// TIA Portal project "Cierre_Centralizado" (V16)

(* hardware
DEVICE "S7-1200 station_1"  S7-1200 Station
   slot 0: "Rack_0"  S7-1200 Rack  Rack  V1.0
   slot 1: "PLC_1"  CPU 1214C AC/DC/Rly  6ES7 214-1BG40-0XB0  V4.2
   slot 3: "AQ 1x12BIT_1"  AQ1 signal board  6ES7 232-4HA30-0XB0  V1.0
*)

// ===== PLC "PLC_1"  CPU 1214C AC/DC/Rly =====

VAR_GLOBAL   // PLC tag table "Entradas"
   "mandoAbrir" AT %I0.0 : Bool;
   "mandoCerrar" AT %I0.1 : Bool;
   "senPC" AT %I0.3 : Bool;
   "senPA" AT %I0.2 : Bool;
   "senVDA" AT %I0.4 : Bool;
   "senVIA" AT %I0.5 : Bool;
   "senVDC" AT %I0.6 : Bool;
   "senVIC" AT %I0.7 : Bool;
END_VAR

VAR_GLOBAL   // PLC tag table "Salidas"
   "releAbrirPuerta" AT %Q0.0 : Bool;
   "releCerrarPuerta" AT %Q0.1 : Bool;
   "releVentanaDerechaAbrir" AT %Q0.2 : Bool;
   "releVentanaIzquierdaAbrir" AT %Q0.3 : Bool;
   "releVentanaDerechaCerrar" AT %Q0.4 : Bool;
   "releVentanaIzquierdaCerrar" AT %Q0.5 : Bool;
END_VAR

VAR_GLOBAL   // PLC tag table "Marcas"
   "mandoAbrir_FA" AT %M6.0 : Bool;
   "mandoCerrar_FA" AT %M6.1 : Bool;
   "mandoCerrar_Aux" AT %M7.1 : Bool;
   "mandoAbrir_Aux" AT %M7.0 : Bool;
END_VAR

DATA_BLOCK "Cierre_Centralizado_DB"   // DB1
{ S7_Optimized_Access := 'TRUE' }
VERSION : 0.1
// stored: InstanceOfName Cierre_Centralizado
"Cierre_Centralizado"
BEGIN
END_DATA_BLOCK

// folder: System blocks/Program resources

DATA_BLOCK "T1"   // DB2
{ S7_Optimized_Access := 'TRUE' }
AUTHOR : Simatic
FAMILY : IEC
NAME : IEC_TMR
VERSION : 1.0
// stored: InstanceOfName IEC_TIMER
"IEC_TIMER"
BEGIN
END_DATA_BLOCK

DATA_BLOCK "T2"   // DB3
{ S7_Optimized_Access := 'TRUE' }
AUTHOR : Simatic
FAMILY : IEC
NAME : IEC_TMR
VERSION : 1.0
// stored: InstanceOfName IEC_TIMER
"IEC_TIMER"
BEGIN
END_DATA_BLOCK

// folder: (top level)

FUNCTION_BLOCK "Cierre_Centralizado"   // FB1, LAD
{ S7_Optimized_Access := 'TRUE' }
VERSION : 0.1
   VAR_INPUT
      Init : Bool := false;
      Reset : Bool;
   END_VAR
   VAR
      X0 : Bool := true;
      X1 : Bool;
      X2 : Bool;
      X3 : Bool;
      X4 : Bool;
      X5 : Bool;
      X6 : Bool;
      X7 : Bool;
      X8 : Bool;
      X9 : Bool;
   END_VAR
BEGIN

REGION Network 1: X0
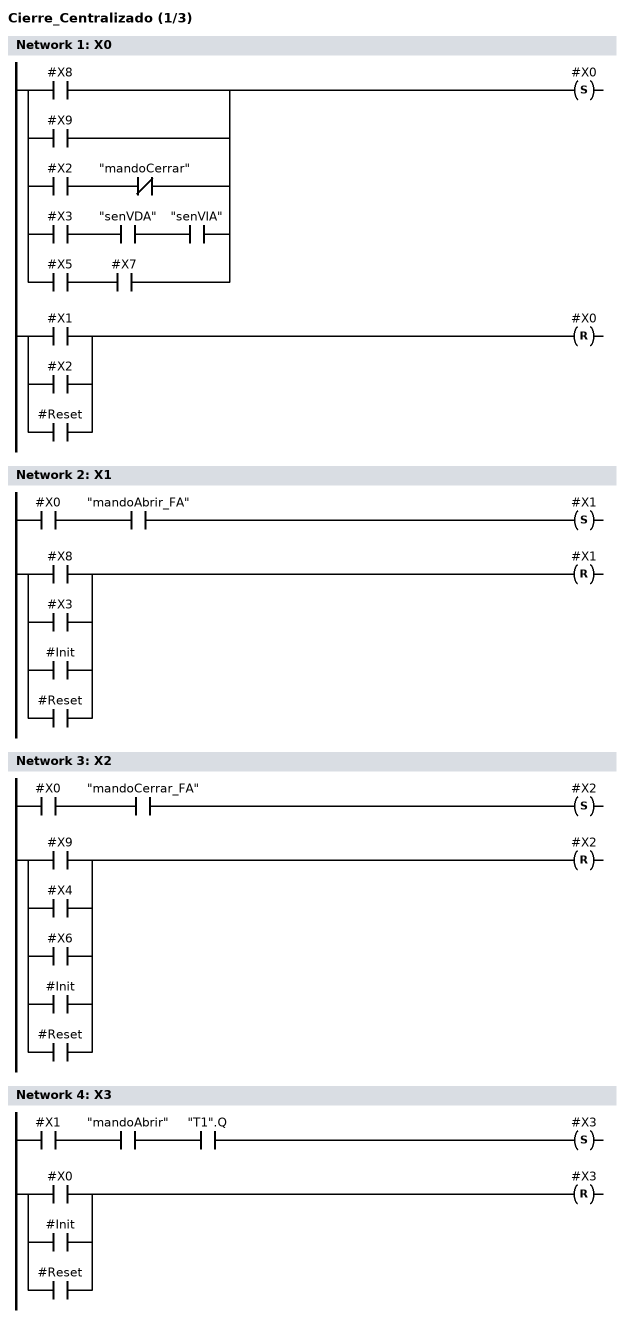
   RUNG wire#powerrail
      Contact( #X8 )
      wire#w1
      S_Coil( #X0 )
   END_RUNG
   RUNG wire#powerrail
      Contact( #X9 )
   END_RUNG wire#w1
   RUNG wire#powerrail
      Contact( #X2 )
      I_Contact( "mandoCerrar" )
   END_RUNG wire#w1
   RUNG wire#powerrail
      Contact( #X3 )
      Contact( "senVDA" )
      Contact( "senVIA" )
   END_RUNG wire#w1
   RUNG wire#powerrail
      Contact( #X5 )
      Contact( #X7 )
   END_RUNG wire#w1
   RUNG wire#powerrail
      Contact( #X1 )
      wire#w2
      R_Coil( #X0 )
   END_RUNG
   RUNG wire#powerrail
      Contact( #X2 )
   END_RUNG wire#w2
   RUNG wire#powerrail
      Contact( #Reset )
   END_RUNG wire#w2
   // the same network as SCL:
   IF #X8 OR #X9 OR (#X2 AND NOT "mandoCerrar") OR (#X3 AND "senVDA" AND "senVIA") OR (#X5 AND #X7) THEN
       #X0 := TRUE;
   END_IF;
   IF #X1 OR #X2 OR #Reset THEN #X0 := FALSE; END_IF;
END_REGION

REGION Network 2: X1
   RUNG wire#powerrail
      Contact( #X0 )
      Contact( "mandoAbrir_FA" )
      S_Coil( #X1 )
   END_RUNG
   RUNG wire#powerrail
      Contact( #X8 )
      wire#w1
      R_Coil( #X1 )
   END_RUNG
   RUNG wire#powerrail
      Contact( #X3 )
   END_RUNG wire#w1
   RUNG wire#powerrail
      Contact( #Init )
   END_RUNG wire#w1
   RUNG wire#powerrail
      Contact( #Reset )
   END_RUNG wire#w1
   // the same network as SCL:
   IF #X0 AND "mandoAbrir_FA" THEN #X1 := TRUE; END_IF;
   IF #X8 OR #X3 OR #Init OR #Reset THEN #X1 := FALSE; END_IF;
END_REGION

REGION Network 3: X2
   RUNG wire#powerrail
      Contact( #X0 )
      Contact( "mandoCerrar_FA" )
      S_Coil( #X2 )
   END_RUNG
   RUNG wire#powerrail
      Contact( #X9 )
      wire#w1
      R_Coil( #X2 )
   END_RUNG
   RUNG wire#powerrail
      Contact( #X4 )
   END_RUNG wire#w1
   RUNG wire#powerrail
      Contact( #X6 )
   END_RUNG wire#w1
   RUNG wire#powerrail
      Contact( #Init )
   END_RUNG wire#w1
   RUNG wire#powerrail
      Contact( #Reset )
   END_RUNG wire#w1
   // the same network as SCL:
   IF #X0 AND "mandoCerrar_FA" THEN #X2 := TRUE; END_IF;
   IF #X9 OR #X4 OR #X6 OR #Init OR #Reset THEN #X2 := FALSE; END_IF;
END_REGION

REGION Network 4: X3
   RUNG wire#powerrail
      Contact( #X1 )
      Contact( "mandoAbrir" )
      Contact( "T1".Q )
      S_Coil( #X3 )
   END_RUNG
   RUNG wire#powerrail
      Contact( #X0 )
      wire#w1
      R_Coil( #X3 )
   END_RUNG
   RUNG wire#powerrail
      Contact( #Init )
   END_RUNG wire#w1
   RUNG wire#powerrail
      Contact( #Reset )
   END_RUNG wire#w1
   // the same network as SCL:
   IF #X1 AND "mandoAbrir" AND "T1".Q THEN #X3 := TRUE; END_IF;
   IF #X0 OR #Init OR #Reset THEN #X3 := FALSE; END_IF;
END_REGION

REGION Network 5: X4
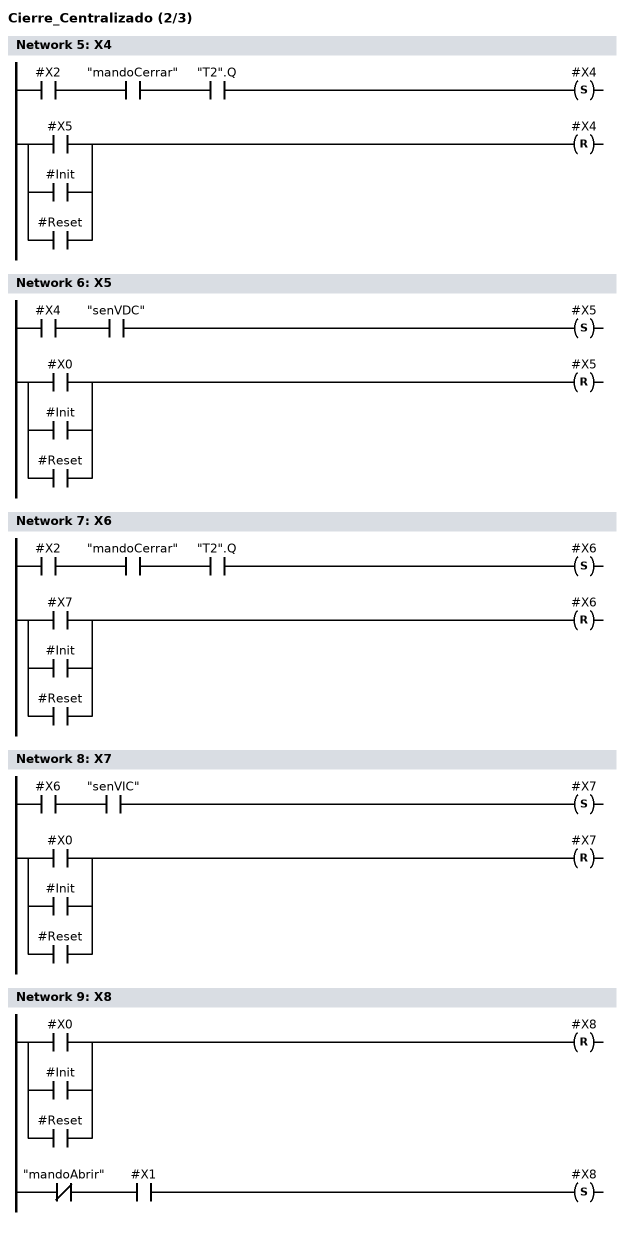
   RUNG wire#powerrail
      Contact( #X2 )
      Contact( "mandoCerrar" )
      Contact( "T2".Q )
      S_Coil( #X4 )
   END_RUNG
   RUNG wire#powerrail
      Contact( #X5 )
      wire#w1
      R_Coil( #X4 )
   END_RUNG
   RUNG wire#powerrail
      Contact( #Init )
   END_RUNG wire#w1
   RUNG wire#powerrail
      Contact( #Reset )
   END_RUNG wire#w1
   // the same network as SCL:
   IF #X2 AND "mandoCerrar" AND "T2".Q THEN #X4 := TRUE; END_IF;
   IF #X5 OR #Init OR #Reset THEN #X4 := FALSE; END_IF;
END_REGION

REGION Network 6: X5
   RUNG wire#powerrail
      Contact( #X4 )
      Contact( "senVDC" )
      S_Coil( #X5 )
   END_RUNG
   RUNG wire#powerrail
      Contact( #X0 )
      wire#w1
      R_Coil( #X5 )
   END_RUNG
   RUNG wire#powerrail
      Contact( #Init )
   END_RUNG wire#w1
   RUNG wire#powerrail
      Contact( #Reset )
   END_RUNG wire#w1
   // the same network as SCL:
   IF #X4 AND "senVDC" THEN #X5 := TRUE; END_IF;
   IF #X0 OR #Init OR #Reset THEN #X5 := FALSE; END_IF;
END_REGION

REGION Network 7: X6
   RUNG wire#powerrail
      Contact( #X2 )
      Contact( "mandoCerrar" )
      Contact( "T2".Q )
      S_Coil( #X6 )
   END_RUNG
   RUNG wire#powerrail
      Contact( #X7 )
      wire#w1
      R_Coil( #X6 )
   END_RUNG
   RUNG wire#powerrail
      Contact( #Init )
   END_RUNG wire#w1
   RUNG wire#powerrail
      Contact( #Reset )
   END_RUNG wire#w1
   // the same network as SCL:
   IF #X2 AND "mandoCerrar" AND "T2".Q THEN #X6 := TRUE; END_IF;
   IF #X7 OR #Init OR #Reset THEN #X6 := FALSE; END_IF;
END_REGION

REGION Network 8: X7
   RUNG wire#powerrail
      Contact( #X6 )
      Contact( "senVIC" )
      S_Coil( #X7 )
   END_RUNG
   RUNG wire#powerrail
      Contact( #X0 )
      wire#w1
      R_Coil( #X7 )
   END_RUNG
   RUNG wire#powerrail
      Contact( #Init )
   END_RUNG wire#w1
   RUNG wire#powerrail
      Contact( #Reset )
   END_RUNG wire#w1
   // the same network as SCL:
   IF #X6 AND "senVIC" THEN #X7 := TRUE; END_IF;
   IF #X0 OR #Init OR #Reset THEN #X7 := FALSE; END_IF;
END_REGION

REGION Network 9: X8
   RUNG wire#powerrail
      Contact( #X0 )
      wire#w1
      R_Coil( #X8 )
   END_RUNG
   RUNG wire#powerrail
      Contact( #Init )
   END_RUNG wire#w1
   RUNG wire#powerrail
      Contact( #Reset )
   END_RUNG wire#w1
   RUNG wire#powerrail
      I_Contact( "mandoAbrir" )
      Contact( #X1 )
      S_Coil( #X8 )
   END_RUNG
   // the same network as SCL:
   IF #X0 OR #Init OR #Reset THEN #X8 := FALSE; END_IF;
   IF NOT "mandoAbrir" AND #X1 THEN #X8 := TRUE; END_IF;
END_REGION

REGION Network 10: X9
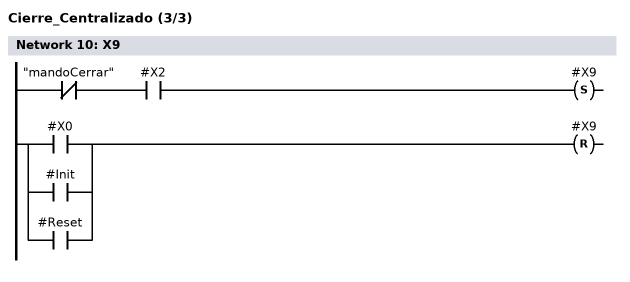
   RUNG wire#powerrail
      I_Contact( "mandoCerrar" )
      Contact( #X2 )
      S_Coil( #X9 )
   END_RUNG
   RUNG wire#powerrail
      Contact( #X0 )
      wire#w1
      R_Coil( #X9 )
   END_RUNG
   RUNG wire#powerrail
      Contact( #Init )
   END_RUNG wire#w1
   RUNG wire#powerrail
      Contact( #Reset )
   END_RUNG wire#w1
   // the same network as SCL:
   IF NOT "mandoCerrar" AND #X2 THEN #X9 := TRUE; END_IF;
   IF #X0 OR #Init OR #Reset THEN #X9 := FALSE; END_IF;
END_REGION
END_FUNCTION_BLOCK

ORGANIZATION_BLOCK "Main"   // OB1, LAD, ProgramCycle
TITLE = "Main Program Sweep (Cycle)"
{ S7_Optimized_Access := 'TRUE' }
VERSION : 0.1
   VAR_INPUT
      Initial_Call : Bool;   // Initial call of this OB
      Remanence : Bool;   // =True, if remanent data are available
   END_VAR
   VAR_TEMP   // added for the SCL form of the ladder/FBD networks
      _w1 : Bool;
      _w2 : Bool;
   END_VAR
BEGIN

REGION Network 1
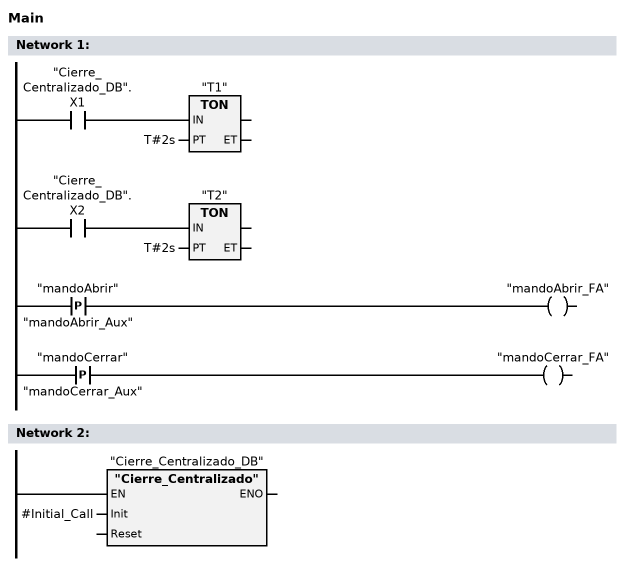
   "T1".TON(IN := "Cierre_Centralizado_DB".X1, PT := T#2s);
   "T2".TON(IN := "Cierre_Centralizado_DB".X2, PT := T#2s);
   #_w1 := "mandoAbrir" AND NOT "mandoAbrir_Aux";   // rising edge of "mandoAbrir"
   "mandoAbrir_Aux" := "mandoAbrir";
   "mandoAbrir_FA" := #_w1;
   #_w2 := "mandoCerrar" AND NOT "mandoCerrar_Aux";   // rising edge of "mandoCerrar"
   "mandoCerrar_Aux" := "mandoCerrar";
   "mandoCerrar_FA" := #_w2;
END_REGION

REGION Network 2
   RUNG wire#powerrail
      "Cierre_Centralizado_DB"(Init := #Initial_Call, Reset :=)
   END_RUNG
   // the same network as SCL:
   "Cierre_Centralizado_DB"(Init := #Initial_Call);   // "Cierre_Centralizado"
END_REGION
END_ORGANIZATION_BLOCK